TYPE ST_KeyControl :
STRUCT
    Boja  : E_BlinkMarine_Color; // Koju boju želiš
    Blink : BOOL;                // Želiš li da blica
END_STRUCT
END_TYPE

(* stored: Version 1.1.0.1, ProductVersion 3.1.4026.17
   DUT ST_KeyControl: Id {8639a7cd-734c-49f0-8afc-10ffc81be459} *)
